{attribute addProperty BoxType "EK1100-0000-0018"}
{attribute addProperty Id "Beckhoff_EL19xxEK1122Beckhoff_EL19xxEK1122_DE3ACA7D162A_0001_EL1918_0000_0016EL1918_BB8AB34720225.25"}
{attribute addProperty CRC "966825071"}
{attribute addProperty SizeInBites "218"}
{attribute addProperty SizeInBytes "27.25"}
TYPE Beckhoff_EL19xx_39A0946F EXTENDS EK1100_179A0949 :
STRUCT
	{attribute addProperty Name "Beckhoff_EL19xxEK1122"}
	Beckhoff_EL19xxEK1122 : Beckhoff_EL19xxEK1122_DE3ACA7D;
	{attribute addProperty Name "A_0001_EL1918_0000_0016"}
	A_0001_EL1918_0000_0016 : EL1918_BB8AB347;
END_STRUCT
END_TYPE

(* stored: Version 1.2.0.0, ProductVersion 3.1.4024.9
   DUT Beckhoff_EL19xx_39A0946F: Id {c35b2cc9-afba-4c5c-9ea7-3bcad5d7d565} *)
